RoboDK station: kuka_station.rdk

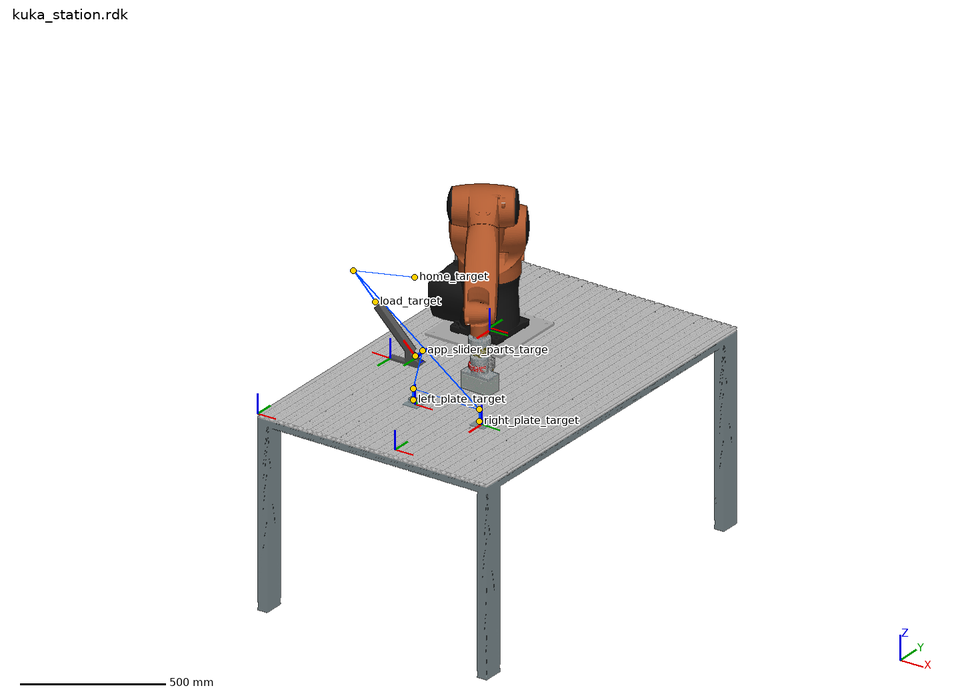
[picture v0: the station drawn from its stored meshes, robots at their saved joint values, targets as dots, program paths as lines]
Station kuka_station (saved by RoboDK 5.5.2). Poses are relative to the parent item; angles as X-Y-Z fixed-axis rotations.
  - frame table_frame at (0, 0, 0) mm
    - object table_object at (0, 0, 0) mm, size 960.1 x 1500 x 750 mm, geometry from table_object.sld
    - frame base_plate_frame at (280, 990, 0) mm, rotated rx 0 ry 0 rz -90 deg
      - object base_plate_object at (0, 0, 0) mm, size 320 x 320 x 10 mm, geometry from base_plate_object.sld
    - frame slider_frame at (125, 617, 0) mm, rotated rx 0 ry 0 rz 180 deg
      - object slider_object at (0, 0, 0) mm, size 198.7 x 26 x 198.7 mm, 1 curves, geometry from slider_object.sld
    - frame slider_parts_frame at (232.7, 617, 30.7) mm, rotated rx 0 ry -45 rz 180 deg
    - frame pick_and_drop_frame at (550, 37, 0) mm
    - frame right_frame at (680, 370, 0) mm, rotated rx 0 ry 0 rz -90 deg
      - object right_plate_object at (0, 0, 0) mm, size 60 x 60 x 9 mm, 1 curves, geometry from right_plate_object.sld
    - frame left_frame at (400, 370, 0) mm
      - object left_plate_object at (0, 0, 0) mm, size 60 x 60 x 9 mm, 1 curves, geometry from left_plate_object.sld
    - frame kuka_frame at (280, 990, 10) mm
      - robot KUKA KR 6 R900 sixx: 6 axes, payload 6 kg, reach 901 mm, repeatability 0.03 mm, weight 52 kg
          modified DH rows (alpha deg, a mm, theta deg, d mm): 0, 0, 0, 400; -90, 25, 0, 0; 0, 455, -90, 0; -90, 35, 0, 420; 90, 0, 0, 0; -90, 0, 180, 80
          joint limits [-170, -190, -120, -185, -120, -350] to [170, 45, 156, 185, 120, 350]; home [0, -90, 90, 0, 0, 0]; saved at [57.686, -34.913, 74.855, -180, -50.058, 192.686]
        - robot gripper: 1 axes
            joint limits [0] to [50]; home [0]; saved at [50]
        - tool gripper_TCP, TCP at (0, 0, 288) mm, rotated rx 0 ry 0 rz 45 deg
    - target home_target (Cartesian target) at (399.96, 369.99, 484.97) mm, rotated rx 180 ry 0 rz 0 deg; joints [74.05, -39.88, 97.01, -180, -32.87, 122.05] of KUKA KR 6 R900 sixx
    - target left_plate_target (Cartesian target) at (393.5, 370, 14.5) mm, rotated rx -180 ry 0 rz 0 deg; joints [79.626, -41.412, 97.379, -180, -34.033, 124.626] of KUKA KR 6 R900 sixx
    - target app_left_plate_target (Cartesian target) at (393.5, 370, 57.5) mm, rotated rx -180 ry 0 rz 0 deg; joints [79.626, -45.516, 97.456, -180, -38.06, 124.626] of KUKA KR 6 R900 sixx
    - target right_plate_target (Cartesian target) at (676.96, 362.41, 14.6) mm, rotated rx 180 ry 0 rz 90 deg; joints [57.686, -31.288, 74.784, -180, -46.504, 192.686] of KUKA KR 6 R900 sixx
    - target app_right_plate_target (Cartesian target) at (676.96, 362.41, 59.6) mm, rotated rx 180 ry 0 rz 90 deg; joints [57.686, -34.913, 74.855, -180, -50.058, 192.686] of KUKA KR 6 R900 sixx
    - target app_slider_parts_target (Cartesian target) at (260.28, 617, 66.76) mm, rotated rx 180 ry 45 rz 0 deg; joints [57.188, -45.773, 126.609, -129.557, -50.427, 55] of KUKA KR 6 R900 sixx
    - target slider_parts_target (Cartesian target) at (229.87, 617, 36.36) mm, rotated rx -180 ry 45 rz 0 deg; joints [60.61, -41.783, 127.838, -122.654, -47.034, 49.699] of KUKA KR 6 R900 sixx
    - target load_target (Cartesian target) at (63.12, 616.34, 197.75) mm, rotated rx -179.98 ry 44.81 rz 0 deg; joints [83.518, -69.18, 137.228, -115.856, -51.087, 73.532] of KUKA KR 6 R900 sixx
    - target app_load_target (Cartesian target) at (-29.33, 617, 291.33) mm, rotated rx 180 ry 45 rz 0 deg; joints [97.501, -81.855, 133.744, -117.425, -52.169, 93.78] of KUKA KR 6 R900 sixx
    - target close_gripper_target (joint target) at (-29.33, 617, 291.33) mm, rotated rx 180 ry 45 rz 0 deg; joints [20, -81.855, 133.744, -117.425, -52.169, 93.78] of gripper
    - target open_gripper_target (joint target) at (-144.59, 617, -0.71) mm, rotated rx 145.71 ry 31.14 rz -52.83 deg; joints [50] of gripper
  - folder programs
    - program factory_reset (1 instructions, listed below)
    - program close_gripper (3 instructions, listed below)
    - program open_gripper (3 instructions, listed below)
    - program main (31 instructions, listed below)
  - object part_object at (399.92, 370, 11.51) mm, rotated rx 0 ry 0 rz -180 deg, size 40 x 20 x 20 mm, 1 curves, geometry from part_object.sld
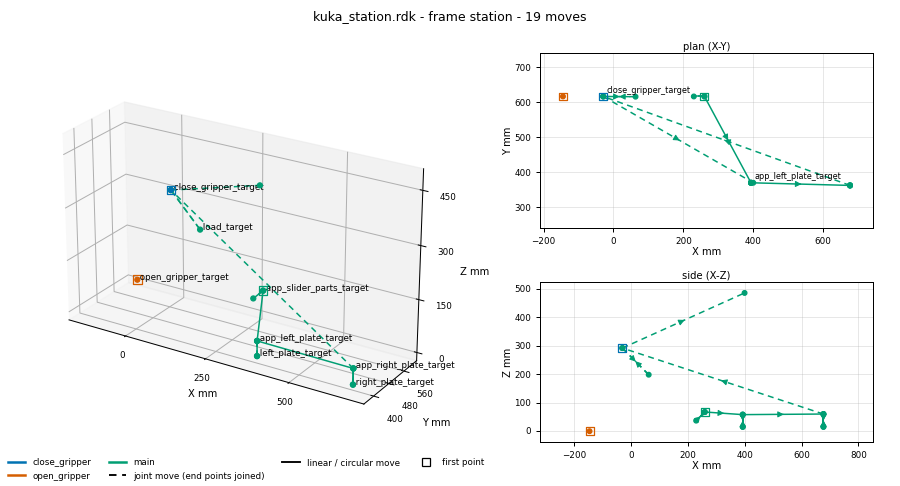
[picture p0: tool path of kuka_station.rdk in frame station, 19 of 19 moves have a stored position in this frame; points joined in program order, loops and branches not executed]

--- program factory_reset (robot KUKA KR 6 R900 sixx) ---
  Replace objects

--- program close_gripper (robot gripper) ---
  Set Ref.: table_frame
  Set Tool: gripper_TCP
  MoveJ (close_gripper_target)

--- program open_gripper (robot gripper) ---
  Set Ref.: table_frame
  Set Tool: gripper_TCP
  MoveJ (open_gripper_target)

--- program main (robot KUKA KR 6 R900 sixx) ---
  Set Ref.: table_frame
  Set Tool: gripper_TCP
  MoveJ (app_slider_parts_target)
  MoveJ (slider_parts_target)
  Call close_gripper
  Attach to gripper_TCP
  MoveL (app_slider_parts_target)
  MoveL (app_left_plate_target)
  MoveJ (left_plate_target)
  Call open_gripper
  Detach from gripper_TCP
  MoveL (app_left_plate_target)
  MoveJ (left_plate_target)
  Call close_gripper
  Attach to gripper_TCP
  MoveJ (app_left_plate_target)
  MoveL (app_right_plate_target)
  MoveL (right_plate_target)
  Call open_gripper
  Detach from gripper_TCP
  MoveL (app_right_plate_target)
  MoveL (right_plate_target)
  Call close_gripper
  Attach to gripper_TCP
  MoveJ (app_right_plate_target)
  MoveJ (app_load_target)
  MoveJ (load_target)
  Call open_gripper
  Detach from gripper_TCP
  MoveJ (app_load_target)
  MoveJ (home_target)
